FUNCTION_BLOCK Sensor_Nivel_4a20 (* Composite Function Block Type *)
  (* Standard: 61499-2 *)
  (* Version 0.0, 2/9/2026, Schneider Electric, template *)
  PACKAGE Hidryco.HidrycoLib;
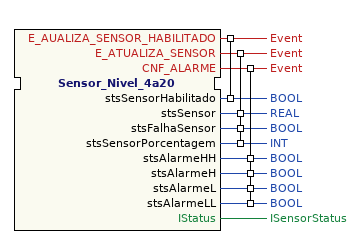
  EVENT_OUTPUT
    E_AUALIZA_SENSOR_HABILITADO WITH stsSensorHabilitado;
    E_ATUALIZA_SENSOR WITH stsSensor, stsFalhaSensor, stsSensorPorcentagem;
    CNF_ALARME WITH stsAlarmeHH, stsAlarmeH, stsAlarmeL, stsAlarmeLL;
  END_EVENT
  VAR_OUTPUT
    stsSensorHabilitado : BOOL;
    stsSensor : REAL;
    stsFalhaSensor : BOOL;
    stsSensorPorcentagem : INT;
    stsAlarmeHH : BOOL;
    stsAlarmeH : BOOL;
    stsAlarmeL : BOOL;
    stsAlarmeLL : BOOL;
  END_VAR
  PLUGS
    IStatus : ISensorStatus;
  END_PLUGS
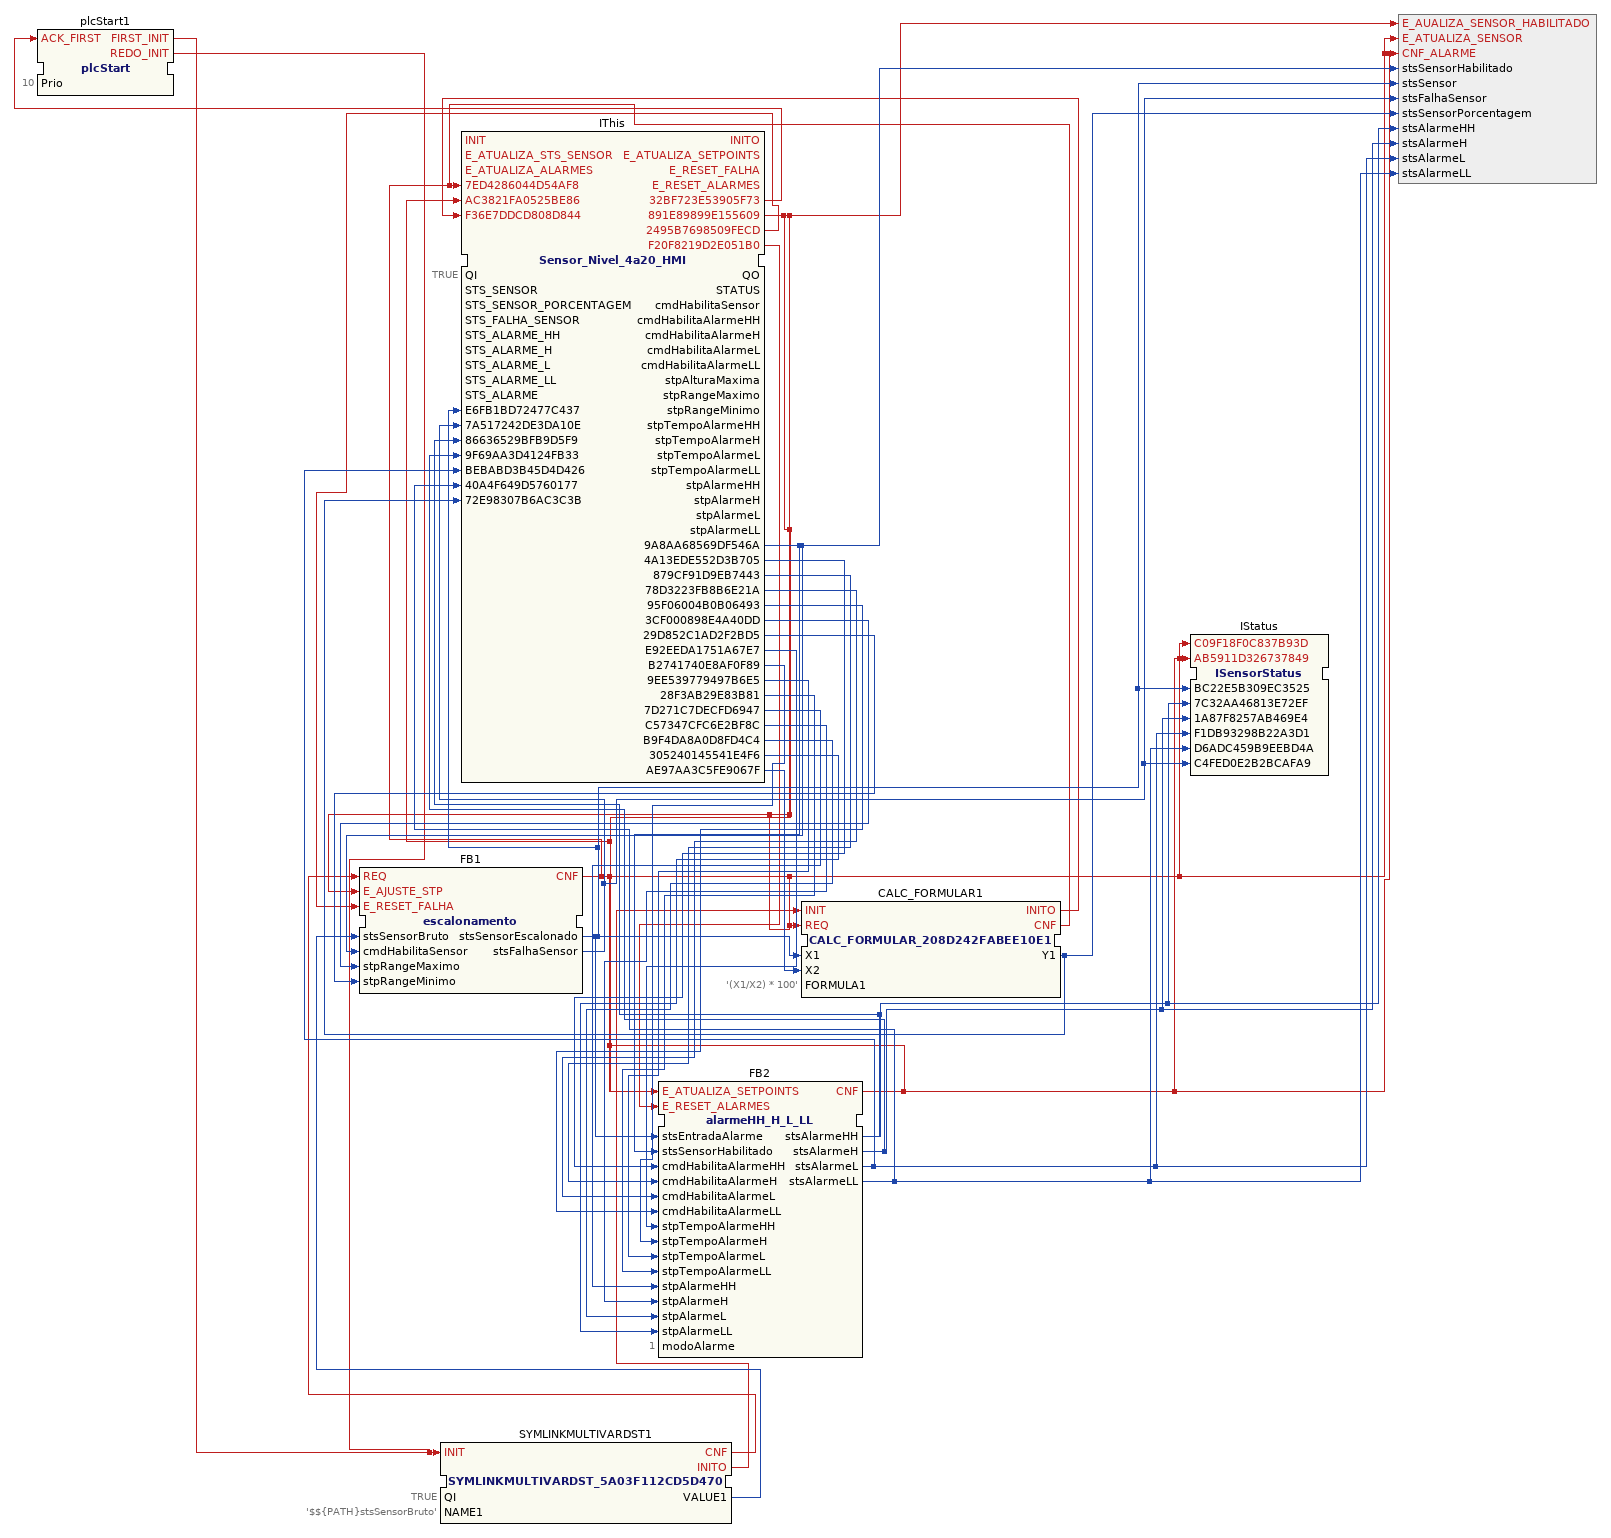
  (* 0 - INITIALIZATION *)
  (* 1 - FUNCTIONAL INPUT INTERFACE *)
  (* 6 - OT-IT INTERFACE *)
  (* 2 - FUNCTIONAL OUTPUT INTERFACE *)
  (* 3 - FIELD INTERFACE *)
  (* 5 - LOGICS *)
  (* 5.B - OPERATION MODE MANAGEMENT *)
  (* 5.C - INTERLOCKS MANAGEMENT *)
  (* 5.A - FUNCTIONAL BEHAVIORS *)
  FBS
    FB1 : escalonamento;
    FB2 : alarmeHH_H_L_LL(modoAlarme := 1);
    IThis : Sensor_Nivel_4a20_HMI(QI := TRUE);
    CALC_FORMULAR1 : CALC_FORMULAR_208D242FABEE10E1(FORMULA1 := '(X1/X2) * 100'); {SET_ATTRIBUTE(Configuration.GenericFBType.InterfaceParams, Runtime.Standard#OUTCNT:=1;INCNT:=2;X${INCNT$}:REAL,REAL;Y${OUTCNT$}:INT)}
    plcStart1 : plcStart(Prio := 10);
    SYMLINKMULTIVARDST1 : SYMLINKMULTIVARDST_5A03F112CD5D470(QI := TRUE, NAME1 := '$${PATH}stsSensorBruto'); {SET_ATTRIBUTE(Configuration.GenericFBType.InterfaceParams, Runtime.System#I:=1;VALUE${I$}:INT)}
  END_FBS
  EVENT_CONNECTIONS
    SYMLINKMULTIVARDST1.CNF TO FB1.REQ;
    FB1.CNF TO E_ATUALIZA_SENSOR;
    FB1.CNF TO FB2.E_ATUALIZA_SETPOINTS;
    plcStart1.FIRST_INIT TO SYMLINKMULTIVARDST1.INIT;
    plcStart1.REDO_INIT TO SYMLINKMULTIVARDST1.INIT;
    FB1.CNF TO IThis.7ED4286044D54AF8;
    FB2.CNF TO IThis.AC3821FA0525BE86;
    IThis.32BF723E53905F73 TO plcStart1.ACK_FIRST;
    IThis.891E89899E155609 TO FB1.E_AJUSTE_STP;
    IThis.891E89899E155609 TO FB2.E_ATUALIZA_SETPOINTS;
    IThis.891E89899E155609 TO E_AUALIZA_SENSOR_HABILITADO;
    IThis.2495B7698509FECD TO FB1.E_RESET_FALHA;
    IThis.F20F8219D2E051B0 TO FB2.E_RESET_ALARMES;
    SYMLINKMULTIVARDST1.INITO TO CALC_FORMULAR1.INIT;
    FB1.CNF TO CALC_FORMULAR1.REQ;
    IThis.891E89899E155609 TO CALC_FORMULAR1.REQ;
    CALC_FORMULAR1.INITO TO IThis.F36E7DDCD808D844;
    CALC_FORMULAR1.CNF TO IThis.7ED4286044D54AF8;
    FB2.CNF TO CNF_ALARME;
    FB1.CNF TO IStatus.C09F18F0C837B93D;
    FB2.CNF TO IStatus.AB5911D326737849;
    FB1.CNF TO IStatus.AB5911D326737849;
  END_CONNECTIONS
  DATA_CONNECTIONS
    SYMLINKMULTIVARDST1.VALUE1 TO FB1.stsSensorBruto;
    FB1.stsSensorEscalonado TO FB2.stsEntradaAlarme;
    FB1.stsFalhaSensor TO stsFalhaSensor;
    FB1.stsSensorEscalonado TO stsSensor;
    FB1.stsSensorEscalonado TO IThis.E6FB1BD72477C437;
    FB1.stsFalhaSensor TO IThis.7A517242DE3DA10E;
    FB2.stsAlarmeHH TO IThis.86636529BFB9D5F9;
    FB2.stsAlarmeH TO IThis.9F69AA3D4124FB33;
    FB2.stsAlarmeL TO IThis.BEBABD3B45D4D426;
    FB2.stsAlarmeLL TO IThis.40A4F649D5760177;
    IThis.9A8AA68569DF546A TO FB1.cmdHabilitaSensor;
    IThis.9A8AA68569DF546A TO FB2.stsSensorHabilitado;
    IThis.9A8AA68569DF546A TO stsSensorHabilitado;
    IThis.4A13EDE552D3B705 TO FB2.cmdHabilitaAlarmeHH;
    IThis.879CF91D9EB7443 TO FB2.cmdHabilitaAlarmeH;
    IThis.78D3223FB8B6E21A TO FB2.cmdHabilitaAlarmeL;
    IThis.95F06004B0B06493 TO FB2.cmdHabilitaAlarmeLL;
    IThis.3CF000898E4A40DD TO FB1.stpRangeMaximo;
    IThis.29D852C1AD2F2BD5 TO FB1.stpRangeMinimo;
    IThis.E92EEDA1751A67E7 TO FB2.stpTempoAlarmeHH;
    IThis.B2741740E8AF0F89 TO FB2.stpTempoAlarmeH;
    IThis.9EE539779497B6E5 TO FB2.stpTempoAlarmeL;
    IThis.28F3AB29E83B81 TO FB2.stpTempoAlarmeLL;
    IThis.7D271C7DECFD6947 TO FB2.stpAlarmeHH;
    IThis.C57347CFC6E2BF8C TO FB2.stpAlarmeH;
    IThis.B9F4DA8A0D8FD4C4 TO FB2.stpAlarmeL;
    IThis.305240145541E4F6 TO FB2.stpAlarmeLL;
    FB1.stsSensorEscalonado TO CALC_FORMULAR1.X1;
    IThis.AE97AA3C5FE9067F TO CALC_FORMULAR1.X2;
    CALC_FORMULAR1.Y1 TO IThis.72E98307B6AC3C3B;
    CALC_FORMULAR1.Y1 TO stsSensorPorcentagem;
    FB2.stsAlarmeHH TO stsAlarmeHH;
    FB2.stsAlarmeH TO stsAlarmeH;
    FB2.stsAlarmeL TO stsAlarmeL;
    FB2.stsAlarmeLL TO stsAlarmeLL;
    FB1.stsSensorEscalonado TO IStatus.BC22E5B309EC3525;
    FB2.stsAlarmeHH TO IStatus.7C32AA46813E72EF;
    FB2.stsAlarmeH TO IStatus.1A87F8257AB469E4;
    FB2.stsAlarmeL TO IStatus.F1DB93298B22A3D1;
    FB2.stsAlarmeLL TO IStatus.D6ADC459B9EEBD4A;
    FB1.stsFalhaSensor TO IStatus.C4FED0E2B2BCAFA9;
  END_CONNECTIONS
END_FUNCTION_BLOCK
